Yaskawa INFORM job: GO-TO-STATION-1-BACK.JBI

/JOB
//NAME GO-TO-STATION-1-BACK
//POS
///NPOS 2,0,0,1,0,0
///TOOL 0
///POSTYPE PULSE
///PULSE
C00000=-316465,-222014,-26224,0,-132993,0
C00001=-315020,-58346,-62489,-105692,-50880,109304
P00000=0,-222014,-26224,0,-132993,0
//INST
///DATE 2018/08/27 13:55
///ATTR SC,RW
///GROUP1 RB1
NOP
MOVJ P0000 VJ=50.00
'*****
SETREG MREG#(1) 1
MOVJ C00000 VJ=25.00
'*****
SETREG MREG#(1) 20
MOVJ C00001 VJ=25.00
'*****
SETREG MREG#(1) 21
END
